TYPE "PLCtoMES_AlarmExchange"
VERSION : 0.1
   STRUCT
      "P-Alarm[X]" : Array[1..1024] of Bool;
      Reserve : Array[1..872] of Byte;
   END_STRUCT;

END_TYPE

